// Mitsubishi GX Works2 project: teST   PLC: Q26UDV

PROGRAM MAIN
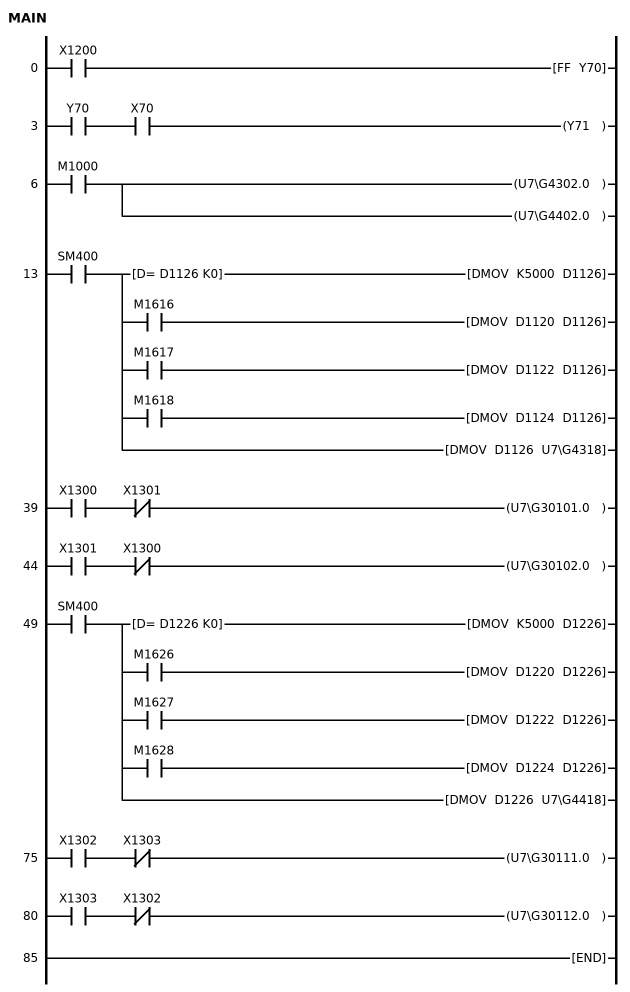
0     LD      X1200
      FF      Y70
3     LD      Y70
      AND     X70
      OUT     Y71
6     LD      M1000
      OUT     U7\G4302.0
      OUT     U7\G4402.0
13    LD      SM400
      MPS
      ANDD=   D1126 K0
      DMOV    K5000 D1126
      MRD
      AND     M1616
      DMOV    D1120 D1126
      MRD
      AND     M1617
      DMOV    D1122 D1126
      MRD
      AND     M1618
      DMOV    D1124 D1126
      MPP
      DMOV    D1126 U7\G4318
39    LD      X1300
      ANI     X1301
      OUT     U7\G30101.0
44    LD      X1301
      ANI     X1300
      OUT     U7\G30102.0
49    LD      SM400
      MPS
      ANDD=   D1226 K0
      DMOV    K5000 D1226
      MRD
      AND     M1626
      DMOV    D1220 D1226
      MRD
      AND     M1627
      DMOV    D1222 D1226
      MRD
      AND     M1628
      DMOV    D1224 D1226
      MPP
      DMOV    D1226 U7\G4418
75    LD      X1302
      ANI     X1303
      OUT     U7\G30111.0
80    LD      X1303
      ANI     X1302
      OUT     U7\G30112.0
85    END
END_PROGRAM

PROGRAM HMI
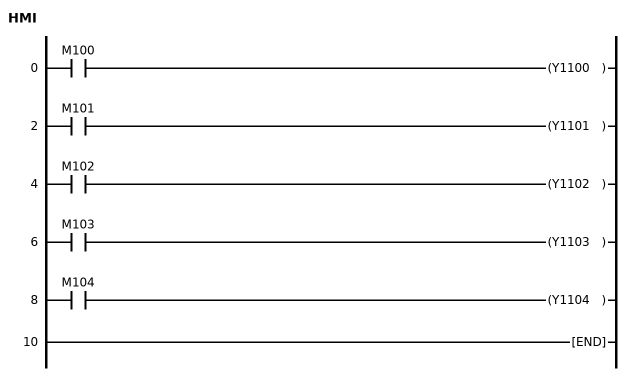
0     LD      M100
      OUT     Y1100
2     LD      M101
      OUT     Y1101
4     LD      M102
      OUT     Y1102
6     LD      M103
      OUT     Y1103
8     LD      M104
      OUT     Y1104
10    END
END_PROGRAM

PROGRAM INPUT
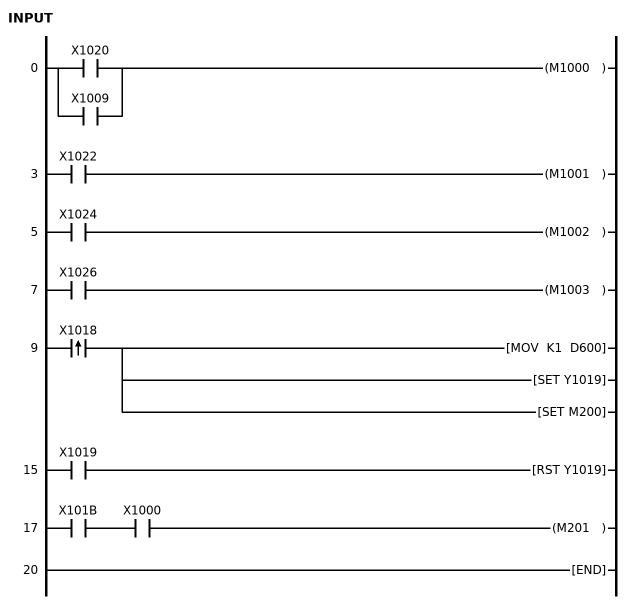
0     LD      X1020
      OR      X1009
      OUT     M1000
3     LD      X1022
      OUT     M1001
5     LD      X1024
      OUT     M1002
7     LD      X1026
      OUT     M1003
9     LDP     X1018
      MOV     K1 D600
      SET     Y1019
      SET     M200
15    LD      X1019
      RST     Y1019
17    LD      X101B
      AND     X1000
      OUT     M201
20    END
END_PROGRAM
